Staubli VAL3: onExit.pgx

program onExit()
begin
  //
  //  Kill everything
  logMsg("[VALlaser] INTERFACE:Quit")
  use:nToSuperV=1
  //
  //
end
